(* PLC project Generated.project, CODESYS CODESYS V3.5 SP19 Patch 1 *)
(* stored: creationDateTime 2026-09-02T08:09:19.557899, modificationDateTime 2026-09-02T08:09:19.557899 *)

(* ======================================================================= 🧩 ST_Fault — Brique socle défaut (2 vues : live + latchée) ─────────────────────────────────────────────────────────────── 🎯 Rôle : porter l'état défaut d'un composant, applicable dans TOUS les cas (acquittable ou non), sans brique warning séparée. • Vue LIVE (Error / ErrorId) : suit la cause, retombe seule à 0. • Vue LATCHÉE (Latched / LatchedId): mémorisée au défaut, reste jusqu'au front Reset. Le choix acquittable / non-acquittable se fait PAR CAUSE (ST_FaultCause.Latching), jamais par bloc. 🔒 Sécurité : interlock TOUJOURS sur la cause brute (Error / ErrorId), jamais sur l'acquittement. Reset TOUJOURS effectif, jamais conditionné (std §9). 🧬 Composition : brique de base réutilisable — sortie de FB, struct métier, GVL. Texte IHM NON stocké ici : dérivé côté IHM depuis LatchedId / ErrorId. 📄 Doc : DOC/STDS/CODE_QUALITY_STANDARDS.md §2quinquies / §9 ======================================================================= *)
TYPE ST_Fault : STRUCT
  Error : BOOL;  (* <-- [DIAG] vue LIVE : au moins une cause présente maintenant *)
  ErrorId : WORD;  (* <-- [DIAG] bitfield des causes présentes maintenant (0 si aucune) *)
  Latched : BOOL;  (* <-- [DIAG] vue LATCHÉE : défaut non acquitté, reste jusqu'au front Reset *)
  LatchedId : WORD;  (* <-- [DIAG] ErrorId figé à l'apparition du défaut, effacé au Reset *)
END_STRUCT;
END_TYPE

(* ======================================================================= 🧩 ST_FaultCause — Cause élémentaire alimentant ST_Fault (socle FB_FaultCore) ─────────────────────────────────────────────────────────────── 🎯 Rôle : une cause exprimée EN CLAIR (BOOL + libellé), sans bitfield ni masque. Le FB métier remplit une liste (ARRAY[0..15] OF ST_FaultCause) ; le socle FB_FaultCore en déduit ST_Fault (vue live + vue latchée). 🔒 Sécurité : interlock TOUJOURS sur Active (cause brute), jamais sur le latch. Latching = TRUE → la cause ARME la vue latchée (défaut à acquitter). Latching = FALSE → la cause n'alimente que la vue live (retombe seule). Fail-safe : une cause laissée à Latching=FALSE reste visible en live — pour la rendre acquittable, il faut le déclarer explicitement. 📄 Doc : DOC/STDS/CODE_QUALITY_STANDARDS.md §2quinquies / §9 ======================================================================= *)
TYPE ST_FaultCause : STRUCT
  Active : BOOL;  (* 1 = cause présente maintenant (interlock sur cette valeur) *)
  Latching : BOOL;  (* 1 = cause à acquitter (arme Latched) ; 0 = live seulement *)
  Texte : STRING;  (* libellé prêt IHM (non stocké dans ST_Fault, dérivé côté IHM) *)
END_STRUCT;
END_TYPE

(* ======================================================================= 🧩 ST_Lifecycle — Brique socle cycle d'exécution ─────────────────────────────────────────────────────────────── 🎯 Rôle : porter l'avancement d'une action à cycle (organe, séquenceur). Optionnelle : un FB purement synchrone (conditionneur, filtre, joystick) ne la porte pas. 🧬 Composition : brique de base réutilisable, composée avec ST_Fault. 📄 Doc : DOC/STDS/CODE_QUALITY_STANDARDS.md §2quinquies ======================================================================= *)
TYPE ST_Lifecycle : STRUCT
  Busy : BOOL;  (* <-- [STAT] 1 = action en cours *)
  Done : BOOL;  (* <-- [STAT] 1 = action terminée avec succès *)
END_STRUCT;
END_TYPE

(* ═══════════════════════════════════════════════════════════════ ⚙️ FB_Recover_Ethercat — Relance à chaud du maître EtherCAT ─────────────────────────────────────────────────────────────── 🎯 Rôle : sur front Request, machine à l'arrêt, attend une tempo power-up puis émet RestartPulse (→ EtherCAT_Master.xRestart, piloté par PRG_02) et surveille xConfigFinished / xError jusqu'au retour du bus. 🔒 Sécurité : ne relance aucun mouvement ; RestartPulse conditionné MachineStopped ; InvalidateEncoders force le re-référencement à la reprise. 📄 Doc métier : DOC/AF/AF_Partie-12_Fonction_Diagnostic_v1.4.md ═══════════════════════════════════════════════════════════════ *)
FUNCTION_BLOCK FB_Recover_Ethercat
  VAR_INPUT
    Enable : BOOL;  (* === CONTRAT STANDARD (Enable + Reset) === --> [CMD] Autorisation generale *)
    Reset : BOOL;  (* --> [CMD] Front acquittement defauts *)
    Request : BOOL;  (* === COMMANDES === --> [CMD] Front = demande de relance (= FaultMachineReset_IHM si bus en erreur) *)
    BusInError : BOOL;  (* --> [HW] TRUE = au moins un esclave EtherCAT hors RUNNING OU maitre en erreur *)
    MasterConfigFinished : BOOL;  (* === RETOURS MAITRE ETHERCAT (cables depuis PRG_02 : EtherCAT_Master.* ) === --> [HW] EtherCAT_Master.xConfigFinished *)
    MasterError : BOOL;  (* --> [HW] EtherCAT_Master.xError *)
    MachineStopped : BOOL;  (* === GARDE SECURITE === --> [SAFE] TRUE = aucun mouvement commande, freins serres *)
    Cfg_PowerUpDelay : TIME := TIME#4s0ms;  (* === REGLAGES === --> [CFG] Delai apres retour energie avant impulsion *)
    Cfg_ConfigTimeout : TIME := TIME#10s0ms;  (* --> [CFG] Delai max attente xConfigFinished *)
  END_VAR
  VAR_OUTPUT
    Ready : BOOL;  (* === CONTRAT STANDARD (Ready + Fault) === <-- [STAT] Surveillance active *)
    Fault : ST_Fault;  (* <-- [DIAG] Defaut (via FB_FaultCore) *)
    Lifecycle : ST_Lifecycle;  (* === CYCLE DE VIE === <-- [STAT] Busy / Done *)
    RestartPulse : BOOL;  (* === SORTIES D'ACTION === <-- [ACT] Impulsion 1 cycle -> EtherCAT_Master.xRestart (piloté par PRG_02) *)
    InvalidateEncoders : BOOL;  (* <-- [ACT] Impulsion a la reprise -> forcer re-homing M1/M2 *)
  END_VAR
  VAR
    instFault : FB_FaultCore;  (* === SOUS-INSTANCES FB === * [INST] Socle defaut *)
    instCauses : ARRAY[0..15] OF ST_FaultCause;  (* . [LOC] Liste des causes en clair *)
    ReqEdge : R_TRIG;  (* === DETECTEURS DE FRONT === . [LOC] Front montant Request *)
    ResetEdge : R_TRIG;  (* . [LOC] Front montant Reset *)
    Step : INT;  (* === MACHINE D'ETAT === . [LOC] 0 IDLE, 1 WAIT_POWERUP, 2 PULSE, 3 WAIT_CONFIG, 4 SETTLE, 5 DONE, 6 FAIL *)
    TonPowerUp : TON;  (* . [LOC] Tempo power-up devices *)
    TonConfig : TON;  (* . [LOC] Timeout attente xConfigFinished *)
    CauseNotStopped : BOOL;  (* === CAUSES (drapeaux latches) === . [LOC] Relance refusee : machine non arretee *)
    CauseConfigTimeout : BOOL;  (* . [LOC] xConfigFinished jamais TRUE dans le delai *)
    CauseMasterError : BOOL;  (* . [LOC] EtherCAT_Master.xError pendant la relance *)
    CauseBusStillDown : BOOL;  (* . [LOC] Relance faite mais esclaves toujours hors RUNNING *)
  END_VAR

            

{region "§1 Gate + fronts + machine d'etat"}
ReqEdge(CLK := Request);
ResetEdge(CLK := Reset);

IF NOT Enable THEN
    Step := 0;
    RestartPulse := FALSE;
    InvalidateEncoders := FALSE;
    Lifecycle.Busy := FALSE;
    Lifecycle.Done := FALSE;
    Ready := FALSE;
    TonPowerUp(IN := FALSE);
    TonConfig(IN := FALSE);
ELSE
    Ready := TRUE;
    RestartPulse := FALSE;      // impulsion : FALSE par defaut, TRUE 1 cycle en step PULSE
    InvalidateEncoders := FALSE;

    // CASE a etiquettes litterales : 0..6 (voir declaration Step).
    CASE Step OF
        0: // IDLE
            Lifecycle.Busy := FALSE;
            TonPowerUp(IN := FALSE);
            TonConfig(IN := FALSE);
            IF ReqEdge.Q AND BusInError THEN
                IF MachineStopped THEN
                    CauseNotStopped    := FALSE;
                    CauseConfigTimeout := FALSE;
                    CauseMasterError   := FALSE;
                    CauseBusStillDown  := FALSE;
                    Lifecycle.Done := FALSE;
                    Step := 1;
                ELSE
                    CauseNotStopped := TRUE; // refus : machine pas a l'arret
                END_IF;
            END_IF;

        1: // WAIT_POWERUP
            Lifecycle.Busy := TRUE;
            TonPowerUp(IN := TRUE, PT := Cfg_PowerUpDelay);
            IF NOT MachineStopped THEN
                CauseNotStopped := TRUE;
                Step := 6;
            ELSIF TonPowerUp.Q THEN
                Step := 2;
            END_IF;

        2: // PULSE
            RestartPulse := TRUE; // 1 cycle -> EtherCAT_Master.xRestart
            Step := 3;

        3: // WAIT_CONFIG
            TonConfig(IN := TRUE, PT := Cfg_ConfigTimeout);
            IF MasterError THEN
                CauseMasterError := TRUE;
                Step := 6;
            ELSIF MasterConfigFinished AND NOT BusInError THEN
                Step := 4;
            ELSIF TonConfig.Q THEN
                IF BusInError THEN
                    CauseBusStillDown := TRUE;
                ELSE
                    CauseConfigTimeout := TRUE;
                END_IF;
                Step := 6;
            END_IF;

        4: // SETTLE
            InvalidateEncoders := TRUE; // 1 cycle -> re-homing obligatoire M1/M2
            Step := 5;

        5: // DONE
            Lifecycle.Busy := FALSE;
            Lifecycle.Done := TRUE;
            IF ReqEdge.Q THEN
                Step := 0; // re-armable
            END_IF;

        6: // FAIL
            Lifecycle.Busy := FALSE;
            IF ResetEdge.Q THEN
                Step := 0;
            END_IF;

        ELSE
            Step := 0;
    END_CASE;
END_IF;
{endregion}

{region "§2 Socle defaut (FB_FaultCore)"}
instCauses[0].Active := CauseNotStopped;    instCauses[0].Latching := TRUE; instCauses[0].Texte := 'Recovery EtherCAT refuse - machine non arretee';
instCauses[1].Active := CauseConfigTimeout; instCauses[1].Latching := TRUE; instCauses[1].Texte := 'Recovery EtherCAT - xConfigFinished timeout';
instCauses[2].Active := CauseMasterError;   instCauses[2].Latching := TRUE; instCauses[2].Texte := 'Recovery EtherCAT - maitre en erreur';
instCauses[3].Active := CauseBusStillDown;  instCauses[3].Latching := TRUE; instCauses[3].Texte := 'Recovery EtherCAT - esclaves hors RUNNING';

instFault(Enable := Enable, Reset := Reset, Causes := instCauses);
Fault := instFault.Fault;
{endregion}

          
END_FUNCTION_BLOCK

(* ======================================================================= 🧩 FB_FaultCore — Socle de remplissage de ST_Fault (vue live + vue latchée) ─────────────────────────────────────────────────────────────── 🎯 Rôle : à partir d'une LISTE de causes en clair (ARRAY[0..15] OF ST_FaultCause), produire la brique ST_Fault : • Error / ErrorId : vue LIVE, suit les causes Active, retombe seule. • Latched / LatchedId: vue LATCHÉE, chaque bit figé à l'apparition d'une cause `Active AND Latching`, conservé jusqu'au front Reset. 🔒 Sécurité : - interlock TOUJOURS sur `Causes[i].Active` (cause brute), jamais sur le latch. - Reset TOUJOURS effectif, jamais conditionné (std §9) — agit même Enable=FALSE. - Latching=FALSE → cause visible en LIVE seulement (fail-safe : reste visible). - un défaut laté non acquitté reste publié même FB désactivé (pas d'effacement silencieux sur bascule Enable OFF→ON sans Reset). - une cause à acquitter réapparue re-arme son bit (ré-alarme). 🧬 Un seul socle, réutilisé par tout FB `standard` qui expose un ST_Fault. Pas de State, pas de Warning, pas de texte — hors périmètre de ce socle. 📄 Doc : DOC/STDS/CODE_QUALITY_STANDARDS.md §2quinquies / §9 ======================================================================= *)
FUNCTION_BLOCK FB_FaultCore
  VAR_INPUT
    Enable : BOOL;  (* --> [CMD] Autorisation générale du FB porteur *)
    Reset : BOOL;  (* --> [CMD] Front d'acquittement (jamais conditionné, §9) *)
    Causes : ARRAY[0..15] OF ST_FaultCause;  (* --> [CMD] Liste des causes en clair (Active / Latching / Texte) *)
  END_VAR
  VAR_OUTPUT
    Ready : BOOL;  (* <-- [STAT] FB porteur autorisé (= Enable) *)
    Fault : ST_Fault;  (* <-- [DIAG] Brique défaut (mappée 1:1 sur la sortie du FB porteur) *)
  END_VAR
  VAR
    ResetEdge : R_TRIG;  (* . [LOC] Front montant Reset *)
    Latch : ARRAY[0..15] OF BOOL;  (* . [LOC] Bit laté par cause, jusqu'au Reset *)
    i : INT;  (* . [LOC] Index de parcours de la liste *)
  END_VAR

            

{region "§1 Reset (front, toujours effectif)"}
// Front Reset : efface tous les latches. Jamais conditionné, agit même Enable=FALSE (§9).
Ready := Enable;
ResetEdge(CLK := Reset);
IF ResetEdge.Q THEN
    FOR i := 0 TO 15 DO Latch[i] := FALSE; END_FOR;
END_IF;
{endregion}

{region "§2 Vue LIVE — Error / ErrorId"}
// Bitfield des causes présentes MAINTENANT. Retombe seule à 0 quand les causes disparaissent.
// Non évaluée si Enable=FALSE (pas de lecture de cause hors autorisation).
Fault.ErrorId := 0;
IF Enable THEN
    FOR i := 0 TO 15 DO
        IF Causes[i].Active THEN
            Fault.ErrorId := Fault.ErrorId OR SHL(WORD#1, INT_TO_DWORD(i));
        END_IF;
    END_FOR;
END_IF;
Fault.Error := (Fault.ErrorId <> 0);
{endregion}

{region "§3 Armement des latches (causes à acquitter)"}
// Une cause Active ET Latching arme son bit ; le bit reste jusqu'au front Reset (§1),
// même si la cause disparaît. Réapparition => ré-armement (ré-alarme).
IF Enable THEN
    FOR i := 0 TO 15 DO
        IF Causes[i].Active AND Causes[i].Latching THEN
            Latch[i] := TRUE;
        END_IF;
    END_FOR;
END_IF;
{endregion}

{region "§4 Vue LATCHÉE — Latched / LatchedId"}
// Toujours publiée, y compris Enable=FALSE : un défaut non acquitté reste visible.
Fault.LatchedId := 0;
FOR i := 0 TO 15 DO
    IF Latch[i] THEN
        Fault.LatchedId := Fault.LatchedId OR SHL(WORD#1, INT_TO_DWORD(i));
    END_IF;
END_FOR;
Fault.Latched := (Fault.LatchedId <> 0);
{endregion}

          
END_FUNCTION_BLOCK
